{attribute 'qualified_only'}
{attribute 'strict'}
TYPE ENUM_EpicsStatesGeneric :
(
	epics_states_generic_unknown := 0,
	epics_states_generic_in := 1,
	epics_states_generic_out := 2
);
END_TYPE

(* stored: Version 1.1.0.1, ProductVersion 3.1.4022.12
   DUT ENUM_EpicsStatesGeneric: Id {83e92801-70cf-4ab2-9ff0-2f24bad8470e} *)
